{attribute 'linkalways'} 
{attribute 'no_explicit_call' := 'This FB is a CLASS and must be accessed using methods or properties'}
{attribute 'enable_dynamic_creation'}
FUNCTION_BLOCK Node_F_VN_MaxElementElementwise_USINT EXTENDS VisionNode
VAR
    ipContainer : _ITcVnContainer;
    nMax : _USINT(0);
    hrPrev : _HRESULT(S_OK);
    hresult : _HRESULT(S_OK);
END_VAR

METHOD PUBLIC  Clone : I_Node
VAR
	pNode : POINTER TO Node_F_VN_MaxElementElementwise_USINT;
END_VAR
pNode := __NEW(Node_F_VN_MaxElementElementwise_USINT);
Clone := pNode^;
END_METHOD

METHOD FB_init : BOOL
VAR_INPUT
	bInitRetains : BOOL; // if TRUE, the retain variables are initialized (warm start / cold start)
	bInCopyCode : BOOL;  // if TRUE, the instance afterwards gets moved into the copy code (online change)
END_VAR
AddInput('ipContainer', ipContainer);
AddInput('nMax', nMax);
AddInput('hrPrev', hrPrev);
AddOutput('ipContainer', ipContainer);
AddOutput('hresult',hresult);
END_METHOD

METHOD PROTECTED OnExecute : HRESULT
hresult.Value := F_VN_MaxElementElementwise_USINT(
    ipContainer := ipContainer.Value,
    nMax := nMax.Value,
    hrPrev:= hrPrev.Value);
END_METHOD

METHOD PUBLIC PreExecutionCheck
VAR_INPUT
	Check : I_PreExecutionChecks;
END_VAR
Check.IsTrue(ipContainer.IsValid, 'ipContainer must be a valid container');
Check.IsTrue(ipContainer.HasType('CTcVnContainer_Vector_USINT'), 'ipContainer contains incorrect types');
END_METHOD

END_FUNCTION_BLOCK

(* stored: Version 1.1.0.1, ProductVersion 3.1.4024.13
   POU Node_F_VN_MaxElementElementwise_USINT: Id {04e53e23-737c-4dcd-9060-f0849be22213}, SpecialFunc None
   Folder Constructor: Id {23bed7ee-71e6-4f1f-a4c1-b98eb039de9a}
   Method Clone: Id {e0b0eb0d-b2e8-48d0-a098-5a79e76bf254}
   Method FB_init: Id {e39c0b84-aab3-4e5b-a194-3691695df3cd}
   Method OnExecute: Id {43be9ac7-8bcd-4045-9b4c-02866d737be3}
   Method PreExecutionCheck: Id {a28197de-1812-4b2f-a3a1-426eeadc81f0} *)
